(* IEC 61131-3 sources: nana-st/tests/fixtures, 5 files *)

(* ---- chiller.st ---- *)
PROGRAM ChillerControl
VAR_INPUT
    water_temp : REAL;
    high_limit : REAL;
    low_limit : REAL;
END_VAR
VAR_OUTPUT
    chiller_enable : BOOL;
    valve_open : BOOL;
    pump_run : BOOL;
END_VAR

chiller_enable := TRUE;

IF water_temp > high_limit THEN
    valve_open := TRUE;
    pump_run := TRUE;
END_IF;

IF water_temp < low_limit THEN
    valve_open := FALSE;
    pump_run := FALSE;
END_IF;
END_PROGRAM

(* ---- counter.st ---- *)
PROGRAM Counter
VAR
    count : INT := 0;
END_VAR
VAR_OUTPUT
    out : INT;
END_VAR

count := count + 1;
out := count;
END_PROGRAM

(* ---- dosing.st ---- *)
PROGRAM DosingControl
VAR_INPUT
    dosing_mode : INT;
    ph_val : REAL;
    ph_high_limit : REAL;
    ph_low_limit : REAL;
    cond_val : REAL;
    cond_high_limit : REAL;
    cond_low_limit : REAL;
END_VAR
VAR_OUTPUT
    hno3_pump : BOOL;
    naoh_pump : BOOL;
    nano3_pump : BOOL;
END_VAR

IF dosing_mode = 0 THEN
    hno3_pump := FALSE;
    naoh_pump := FALSE;
    nano3_pump := FALSE;

    IF ph_val > ph_high_limit THEN
        hno3_pump := TRUE;
    END_IF;

    IF ph_val < ph_low_limit THEN
        naoh_pump := TRUE;
    END_IF;

    IF cond_val < cond_low_limit THEN
        nano3_pump := TRUE;
    END_IF;

    IF cond_val > cond_high_limit THEN
        nano3_pump := FALSE;
    END_IF;
END_IF;
END_PROGRAM

(* ---- pass_through.st ---- *)
PROGRAM PassThrough
VAR_INPUT
    input : BOOL;
END_VAR
VAR_OUTPUT
    output : BOOL;
END_VAR

output := input;
END_PROGRAM

(* ---- real_branch.st ---- *)
PROGRAM RealBranch
VAR_INPUT
    input : REAL;
END_VAR
VAR
    offset : REAL := 1.5;
END_VAR
VAR_OUTPUT
    output : REAL;
    high : BOOL;
END_VAR

output := input + offset;
high := output >= 10.0;
END_PROGRAM
